// TIA Portal V20 export
VAR_GLOBAL   // PLC tag table "Default tag table"
   BA040AZSDR1_Unwinder1_Interface_AddressIn AT %I5114.0 : "PD_TEL105_IN";
   BA040AZSDR1_Unwinder1_AddressOut AT %Q5114.0 : "PD_TEL105_OUT";
   BA040AZSDR2_Unwinder2_Actor_Interface_AddressIn AT %I5154.0 : "PD_TEL105_IN";
   BA040AZSDR2_Unwinder2_Actor_Interface_AddressOut AT %Q5154.0 : "PD_TEL105_OUT";
   BA040AZSDR5_AnodeMainPnp1AxisX_Actor_Interface_AddressIn AT %I5268.0 : "PD_TEL105_IN";
   BA040AZSDR5_AnodeMainPnp1AxisX_Actor_Interface_AddressOut AT %Q5268.0 : "PD_TEL105_OUT";
   BA040AZSDR6_AnodeMainPnp2AxisX_Actor_Interface_AddressIn AT %I5302.0 : "PD_TEL105_IN";
   BA040AZSDR6_AnodeMainPnp2AxisX_Actor_Interface_AddressOut AT %Q5302.0 : "PD_TEL105_OUT";
   BA040AZSDR7_CathodeMainPnp1AxisX_Actor_Interface_AddressIn AT %I5336.0 : "PD_TEL105_IN";
   BA040AZSDR7_CathodeMainPnp1AxisX_Actor_Interface_AddressOut AT %Q5336.0 : "PD_TEL105_OUT";
   BA040AZSDR8_CathodeMainPnp2AxisX_Actor_Interface_AddressIn AT %I5370.0 : "PD_TEL105_IN";
   BA040AZSDR8_CathodeMainPnp2AxisX_Actor_Interface_AddressOut AT %Q5370.0 : "PD_TEL105_OUT";
   BA040AZSDR9_AnodeMainPnp1AxisY_Actor_Interface_AddressIn AT %I5404.0 : "PD_TEL105_IN";
   BA040AZSDR9_AnodeMainPnp1AxisY_Actor_Interface_AddressOut AT %Q5404.0 : "PD_TEL105_OUT";
   BA040AZSDR10_AnodeMainPnp1AxisZ_Actor_Interface_AddressIn AT %I5438.0 : "PD_TEL105_IN";
   BA040AZSDR10_AnodeMainPnp1AxisZ_Actor_Interface_AddressOut AT %Q5438.0 : "PD_TEL105_OUT";
   BA040AZSDR11_AnodeMainPnp2AxisZ_Actor_Interface_AddressIn AT %I5482.0 : "PD_TEL105_IN";
   BA040AZSDR11_AnodeMainPnp2AxisZ_Actor_Interface_AddressOut AT %Q5482.0 : "PD_TEL105_OUT";
   BA040AZSDR12_CathodeMainPnp2AxisZ_Actor_Interface_AddressIn AT %I5516.0 : "PD_TEL105_IN";
   BA040AZSDR12_CathodeMainPnp2AxisZ_Actor_Interface_AddressOut AT %Q5516.0 : "PD_TEL105_OUT";
   BA040AZSDR13_CathodeMainPnp1AxisX_Actor_Interface_AddressIn AT %I5560.0 : "PD_TEL105_IN";
   BA040AZSDR13_CathodeMainPnp1AxisX_Actor_Interface_AddressOut AT %Q5560.0 : "PD_TEL105_OUT";
   BA040AZSDR14_CathodeMainPnp1AxisZ_Actor_Interface_AddressIn AT %I5604.0 : "PD_TEL105_IN";
   BA040AZSDR14_CathodeMainPnp1AxisZ_Actor_Interface_AddressOut AT %Q5604.0 : "PD_TEL105_OUT";
   BA040AZSDR15_AnodeAlignTableAxisU_Actor_Interface_AddressIn AT %I5648.0 : "PD_TEL105_IN";
   BA040AZSDR15_AnodeAlignTableAxisU_Actor_Interface_AddressOut AT %Q5648.0 : "PD_TEL105_OUT";
   BA040AZSDR16_AnodeAlignTableAxisV_Actor_Interface_AddressIn AT %I5682.0 : "PD_TEL105_IN";
   BA040AZSDR16_AnodeAlignTableAxisV_Actor_Interface_AddressOut AT %Q5682.0 : "PD_TEL105_OUT";
   BA040AZSDR17_AnodeAlignTableAxisW_Actor_Interface_AddressIn AT %I5716.0 : "PD_TEL105_IN";
   BA040AZSDR17_AnodeAlignTableAxisW_Actor_Interface_AddressOut AT %Q5716.0 : "PD_TEL105_OUT";
   BA040AZSDR18_CathodeAlignTableAxisU_Actor_Interface_AddressIn AT %I5750.0 : "PD_TEL105_IN";
   BA040AZSDR18_CathodeAlignTableAxisU_Actor_Interface_AddressOut AT %Q5750.0 : "PD_TEL105_OUT";
   BA040AZSDR19_CathodeAlignTableAxisV_Actor_Interface_AddressIn AT %I5784.0 : "PD_TEL105_IN";
   BA040AZSDR19_CathodeAlignTableAxisV_Actor_Interface_AddressOut AT %Q5784.0 : "PD_TEL105_OUT";
   BA040AZSDR20_CathodeAlignTableAxisW_Actor_Interface_AddressIn AT %I5818.0 : "PD_TEL105_IN";
   BA040AZSDR20_CathodeAlignTableAxisW_Actor_Interface_AddressOut AT %Q5818.0 : "PD_TEL105_OUT";
   BA040AZSDR40_JellyRollWinder1AxisY_Actor_Interface_AddressIn AT %I6588.0 : "PD_TEL105_IN";
   BA040AZSDR40_JellyRollWinder1AxisY_Actor_Interface_AddressOut AT %Q6588.0 : "PD_TEL105_OUT";
   BA040AZSDR41_JellyRollWinder2AxisY_Actor_Interface_AddressIn AT %I6622.0 : "PD_TEL105_IN";
   BA040AZSDR41_JellyRollWinder2AxisY_Actor_Interface_AddressOut AT %Q6622.0 : "PD_TEL105_OUT";
   BA040AZSDR1_UnwinderTopAxisB_Actor_Interface_TorqueDataAddressIn AT %I8000.0 : "PD_TEL750_IN";
   BA040AZSDR1_UnwinderTopAxisB_Actor_Interface_TorqueDataAddressOut AT %Q8000.0 : "PD_TEL750_OUT";
   BA040AZSDR2_UnwinderBottomAxisB_Actor_Interface_TorqueDataAddressIn AT %I8010.0 : "PD_TEL750_IN";
   BA040AZSDR2_UnwinderBottomAxisB_Actor_Interface_TorqueDataAddressOut AT %Q8010.0 : "PD_TEL750_OUT";
   BA040AZSDR4_SepaFeedingRollerAxisB_Actor_Interface_AddressIn AT %I5234.0 : "PD_TEL105_IN";
   BA040AZSDR4_SepaFeedingRollerAxisB_Actor_Interface_AddressOut AT %Q5234.0 : "PD_TEL105_OUT";
   BA040AZSDR4_SepaFeedingRollerAxisB_Actor_Interface_TorqueDataAddressIn AT %I8030.0 : "PD_TEL750_IN";
   BA040AZSDR4_SepaFeedingRollerAxisB_Actor_Interface_TorqueDataAddressOut AT %Q8030.0 : "PD_TEL750_OUT";
   BA040AZSDR21_FinalRollerFrontAxisX_Actor_Interface_AddressIn AT %I5852.0 : "PD_TEL105_IN";
   BA040AZSDR21_FinalRollerFrontAxisX_Actor_Interface_AddressOut AT %Q5852.0 : "PD_TEL105_OUT";
   BA040AZSDR22_FinalRollerRearAxisX_Actor_Interface_AddressIn AT %I5886.0 : "PD_TEL105_IN";
   BA040AZSDR22_FinalRollerRearAxisX_Actor_Interface_AddressOut AT %Q5886.0 : "PD_TEL105_OUT";
   BA040AZSDR23_MendrelAnodeFrontAxisY_Actor_Interface_AddressIn AT %I5920.0 : "PD_TEL105_IN";
   BA040AZSDR23_MendrelAnodeFrontAxisY_Actor_Interface_AddressOut AT %Q5920.0 : "PD_TEL105_OUT";
   BA040AZSDR24_MendrelAnodeFrontAxisZ_Actor_Interface_AddressIn AT %I5954.0 : "PD_TEL105_IN";
   BA040AZSDR24_MendrelAnodeFrontAxisZ_Actor_Interface_AddressOut AT %Q5954.0 : "PD_TEL105_OUT";
   BA040AZSDR25_MendrelAnodeRearAxisY_Actor_Interface_AddressIn AT %I5998.0 : "PD_TEL105_IN";
   BA040AZSDR25_MendrelAnodeRearAxisY_Actor_Interface_AddressOut AT %Q5998.0 : "PD_TEL105_OUT";
   BA040AZSDR26_MendrelAnodeRearAxisZ_Actor_Interface_AddressIn AT %I6032.0 : "PD_TEL105_IN";
   BA040AZSDR26_MendrelAnodeRearAxisZ_Actor_Interface_AddressOut AT %Q6032.0 : "PD_TEL105_OUT";
   BA040AZSDR27_MendrelCathodeFrontAxisY_Actor_Interface_AddressIn AT %I6076.0 : "PD_TEL105_IN";
   BA040AZSDR27_MendrelCathodeFrontAxisY_Actor_Interface_AddressOut AT %Q6076.0 : "PD_TEL105_OUT";
   BA040AZSDR28_MendrelCathodeFrontAxisZ_Actor_Interface_AddressIn AT %I6110.0 : "PD_TEL105_IN";
   BA040AZSDR28_MendrelCathodeFrontAxisZ_Actor_Interface_AddressOut AT %Q6110.0 : "PD_TEL105_OUT";
   BA040AZSDR29_MendrelCathodeRearAxisY_Actor_Interface_AddressIn AT %I6154.0 : "PD_TEL105_IN";
   BA040AZSDR29_MendrelCathodeRearAxisY_Actor_Interface_AddressOut AT %Q6154.0 : "PD_TEL105_OUT";
   BA040AZSDR30_MendrelCathodeRearAxisZ_Actor_Interface_AddressIn AT %I6188.0 : "PD_TEL105_IN";
   BA040AZSDR30_MendrelCathodeRearAxisZ_Actor_Interface_AddressOut AT %Q6188.0 : "PD_TEL105_OUT";
   BA040AZSDR31_StackTableAxisZ_Actor_Interface_AddressIn AT %I6232.0 : "PD_TEL105_IN";
   BA040AZSDR31_StackTableAxisZ_Actor_Interface_AddressOut AT %Q6232.0 : "PD_TEL105_OUT";
   BA040AZSDR32_StackTableOutFrontAxisZ_Actor_Interface_AddressIn AT %I6276.0 : "PD_TEL105_IN";
   BA040AZSDR32_StackTableOutFrontAxisZ_Actor_Interface_AddressOut AT %Q6276.0 : "PD_TEL105_OUT";
   BA040AZSDR33_StackTableOutRearAxisZ_Actor_Interface_AddressIn AT %I6320.0 : "PD_TEL105_IN";
   BA040AZSDR33_StackTableOutRearAxisZ_Actor_Interface_AddressOut AT %Q6320.0 : "PD_TEL105_OUT";
   BA040AZSDR34_SepaClampnCutterAxisX_Actor_Interface_AddressIn AT %I6364.0 : "PD_TEL105_IN";
   BA040AZSDR34_SepaClampnCutterAxisX_Actor_Interface_AddressOut AT %Q6364.0 : "PD_TEL105_OUT";
   BA040AZSDR35_SepaClampnCutterAxisZ_Actor_Interface_AddressIn AT %I6398.0 : "PD_TEL105_IN";
   BA040AZSDR35_SepaClampnCutterAxisZ_Actor_Interface_AddressOut AT %Q6398.0 : "PD_TEL105_OUT";
   BA040AZSDR36_SepaGripperAxisX_Actor_Interface_AddressIn AT %I6442.0 : "PD_TEL105_IN";
   BA040AZSDR36_SepaGripperAxisX_Actor_Interface_AddressOut AT %Q6442.0 : "PD_TEL105_OUT";
   BA040AZSDR37_SepaGripperAxisZ_Actor_Interface_AddressIn AT %I6476.0 : "PD_TEL105_IN";
   BA040AZSDR37_SepaGripperAxisZ_Actor_Interface_AddressOut AT %Q6476.0 : "PD_TEL105_OUT";
   BA040AZSDR38_SepaGripperAxisC_Actor_Interface_AddressIn AT %I6520.0 : "PD_TEL105_IN";
   BA040AZSDR38_SepaGripperAxisC_Actor_Interface_AddressOut AT %Q6520.0 : "PD_TEL105_OUT";
   BA040AZSDR39_JRWinderRearAxisY_Actor_Interface_AddressIn AT %I6554.0 : "PD_TEL105_IN";
   BA040AZSDR39_JRWinderRearAxisY_Actor_Interface_AddressOut AT %Q6554.0 : "PD_TEL105_OUT";
   BA040AZSDR3_CompensatorAxisX_Actor_Interface_AddressIn AT %I5194.0 : "PD_TEL105_IN";
   BA040AZSDR3_CompensatorAxisX_Actor_Interface_AddressOut AT %Q5194.0 : "PD_TEL105_OUT";
   BA040AZSDR3_CompensatorAxisX_Actor_Interface_TorqueDataAddressIn AT %I8020.0 : "PD_TEL750_IN";
   BA040AZSDR3_CompensatorAxisX_Actor_Interface_TorqueDataAddressOut AT %Q8020.0 : "PD_TEL750_OUT";
   BA040AZSDR39_JRWinderRearAxisY_Actor_Interface_TorqueDataAddressIn AT %I8380.0 : "PD_TEL750_IN";
   BA040AZSDR39_JRWinderRearAxisY_Actor_Interface_TorqueDataAddressOut AT %Q8380.0 : "PD_TEL750_OUT";
   BA040AZSDR5_AnodeMainPnp1AxisX_Actor_Interface_TorqueDataAddressIn AT %I8040.0 : "PD_TEL750_IN";
   BA040AZSDR5_AnodeMainPnp1AxisX_Actor_Interface_TorqueDataAddressOut AT %Q8040.0 : "PD_TEL750_OUT";
   BA040AZSDR6_AnodeMainPnp2AxisX_Actor_Interface_TorqueDataAddressIn AT %I8050.0 : "PD_TEL750_IN";
   BA040AZSDR6_AnodeMainPnp2AxisX_Actor_Interface_TorqueDataAddressOut AT %Q8050.0 : "PD_TEL750_OUT";
   BA040AZSDR11_AnodeMainPnp1AxisY_Actor_Interface_TorqueDataAddressIn AT %I8100.0 : "PD_TEL750_IN";
   BA040AZSDR11_AnodeMainPnp1AxisY_Actor_Interface_TorqueDataAddressOut AT %Q8100.0 : "PD_TEL750_OUT";
   BA040AZSDR12_AnodeMainPnp1AxisZ_Actor_Interface_TorqueDataAddressIn AT %I8110.0 : "PD_TEL750_IN";
   BA040AZSDR12_AnodeMainPnp1AxisZ_Actor_Interface_TorqueDataAddressOut AT %Q8110.0 : "PD_TEL750_OUT";
   BA040AZSDR14_AnodeMainPnp2AxisZ_Actor_Interface_TorqueDataAddressIn AT %I8130.0 : "PD_TEL750_IN";
   BA040AZSDR14_AnodeMainPnp2AxisZ_Actor_Interface_TorqueDataAddressOut AT %Q8130.0 : "PD_TEL750_OUT";
   BA040AZSDR15_AnodeAlignTableAxisX_Actor_Interface_TorqueDataAddressIn AT %I8140.0 : "PD_TEL750_IN";
   BA040AZSDR15_AnodeAlignTableAxisX_Actor_Interface_TorqueDataAddressOut AT %Q8140.0 : "PD_TEL750_OUT";
   BA040AZSDR16_AnodeAlignTableAxisY1_Actor_Interface_TorqueDataAddressIn AT %I8150.0 : "PD_TEL750_IN";
   BA040AZSDR16_AnodeAlignTableAxisY1_Actor_Interface_TorqueDataAddressOut AT %Q8150.0 : "PD_TEL750_OUT";
   BA040AZSDR17_AnodeAlignTableAxisY2_Actor_Interface_TorqueDataAddressIn AT %I8160.0 : "PD_TEL750_IN";
   BA040AZSDR17_AnodeAlignTableAxisY2_Actor_Interface_TorqueDataAddressOut AT %Q8160.0 : "PD_TEL750_OUT";
   BA040AZSDR7_CathodeMainPnp1AxisX_Actor_Interface_TorqueDataAddressIn AT %I8060.0 : "PD_TEL750_IN";
   BA040AZSDR7_CathodeMainPnp1AxisX_Actor_Interface_TorqueDataAddressOut AT %Q8060.0 : "PD_TEL750_OUT";
   BA040AZSDR8_CathodeMainPnp2AxisX_Actor_Interface_TorqueDataAddressIn AT %I8070.0 : "PD_TEL750_IN";
   BA040AZSDR8_CathodeMainPnp2AxisX_Actor_Interface_TorqueDataAddressOut AT %Q8070.0 : "PD_TEL750_OUT";
   BA040AZSDR9_CathodeMainPnp1AxisY_Actor_Interface_TorqueDataAddressIn AT %I8080.0 : "PD_TEL750_IN";
   BA040AZSDR9_CathodeMainPnp1AxisY_Actor_Interface_TorqueDataAddressOut AT %Q8080.0 : "PD_TEL750_OUT";
   BA040AZSDR10_CathodeMainPnp1AxisZ_Actor_Interface_TorqueDataAddressIn AT %I8090.0 : "PD_TEL750_IN";
   BA040AZSDR10_CathodeMainPnp1AxisZ_Actor_Interface_TorqueDataAddressOut AT %Q8090.0 : "PD_TEL750_OUT";
   BA040AZSDR13_CathodeMainPnp2AxisZ_Actor_Interface_TorqueDataAddressIn AT %I8120.0 : "PD_TEL750_IN";
   BA040AZSDR13_CathodeMainPnp2AxisZ_Actor_Interface_TorqueDataAddressOut AT %Q8120.0 : "PD_TEL750_OUT";
   BA040AZSDR18_CathodeAlignTableAxisX_Actor_Interface_TorqueDataAddressIn AT %I8170.0 : "PD_TEL750_IN";
   BA040AZSDR18_CathodeAlignTableAxisX_Actor_Interface_TorqueDataAddressOut AT %Q8170.0 : "PD_TEL750_OUT";
   BA040AZSDR19_CathodeAlignTableAxisY1_Actor_Interface_TorqueDataAddressIn AT %I8180.0 : "PD_TEL750_IN";
   BA040AZSDR19_CathodeAlignTableAxisY1_Actor_Interface_TorqueDataAddressOut AT %Q8180.0 : "PD_TEL750_OUT";
   BA040AZSDR20_CathodeAlignTableAxisY2_Actor_Interface_TorqueDataAddressIn AT %I8190.0 : "PD_TEL750_IN";
   BA040AZSDR20_CathodeAlignTableAxisY2_Actor_Interface_TorqueDataAddressOut AT %Q8190.0 : "PD_TEL750_OUT";
   BA040AZSDR21_FinalRollerFrontAxisX_Actor_Interface_TorqueDataAddressIn AT %I8200.0 : "PD_TEL750_IN";
   BA040AZSDR21_FinalRollerFrontAxisX_Actor_Interface_TorqueDataAddressOut AT %Q8200.0 : "PD_TEL750_OUT";
   BA040AZSDR22_FinalRollerRearAxisX_Actor_Interface_TorqueDataAddressIn AT %I8210.0 : "PD_TEL750_IN";
   BA040AZSDR22_FinalRollerRearAxisX_Actor_Interface_TorqueDataAddressOut AT %Q8210.0 : "PD_TEL750_OUT";
   BA040AZSDR23_MendrelAnodeFrontAxisY_Actor_Interface_TorqueDataAddressIn AT %I8220.0 : "PD_TEL750_IN";
   BA040AZSDR23_MendrelAnodeFrontAxisY_Actor_Interface_TorqueDataAddressOut AT %Q8220.0 : "PD_TEL750_OUT";
   BA040AZSDR24_MendrelAnodeFrontAxisZ_Actor_Interface_TorqueDataAddressIn AT %I8230.0 : "PD_TEL750_IN";
   BA040AZSDR24_MendrelAnodeFrontAxisZ_Actor_Interface_TorqueDataAddressOut AT %Q8230.0 : "PD_TEL750_OUT";
   BA040AZSDR25_MendrelAnodeRearAxisY_Actor_Interface_TorqueDataAddressIn AT %I8240.0 : "PD_TEL750_IN";
   BA040AZSDR25_MendrelAnodeRearAxisY_Actor_Interface_TorqueDataAddressOut AT %Q8240.0 : "PD_TEL750_OUT";
   BA040AZSDR26_MendrelAnodeRearAxisZ_Actor_Interface_TorqueDataAddressIn AT %I8250.0 : "PD_TEL750_IN";
   BA040AZSDR26_MendrelAnodeRearAxisZ_Actor_Interface_TorqueDataAddressOut AT %Q8250.0 : "PD_TEL750_OUT";
   BA040AZSDR27_MendrelCathodeFrontAxisY_Actor_Interface_TorqueDataAddressIn AT %I8260.0 : "PD_TEL750_IN";
   BA040AZSDR27_MendrelCathodeFrontAxisY_Actor_Interface_TorqueDataAddressOut AT %Q8260.0 : "PD_TEL750_OUT";
   BA040AZSDR28_MendrelCathodeFrontAxisZ_Actor_Interface_TorqueDataAddressIn AT %I8270.0 : "PD_TEL750_IN";
   BA040AZSDR28_MendrelCathodeFrontAxisZ_Actor_Interface_TorqueDataAddressOut AT %Q8270.0 : "PD_TEL750_OUT";
   BA040AZSDR29_MendrelCathodeRearAxisY_Actor_Interface_TorqueDataAddressIn AT %I8280.0 : "PD_TEL750_IN";
   BA040AZSDR29_MendrelCathodeRearAxisY_Actor_Interface_TorqueDataAddressOut AT %Q8280.0 : "PD_TEL750_OUT";
   BA040AZSDR30_MendrelCathodeRearAxisZ_Actor_Interface_TorqueDataAddressIn AT %I8290.0 : "PD_TEL750_IN";
   BA040AZSDR30_MendrelCathodeRearAxisZ_Actor_Interface_TorqueDataAddressOut AT %Q8290.0 : "PD_TEL750_OUT";
   BA040AZSDR31_StackTableAxisZ_Actor_Interface_TorqueDataAddressIn AT %I8300.0 : "PD_TEL750_IN";
   BA040AZSDR31_StackTableAxisZ_Actor_Interface_TorqueDataAddressOut AT %Q8300.0 : "PD_TEL750_OUT";
   BA040AZSDR32_StackTableOutFrontAxisZ_Actor_Interface_TorqueDataAddressIn AT %I8310.0 : "PD_TEL750_IN";
   BA040AZSDR32_StackTableOutFrontAxisZ_Actor_Interface_TorqueDataAddressOut AT %Q8310.0 : "PD_TEL750_OUT";
   BA040AZSDR33_StackTableOutRearAxisZ_Actor_Interface_TorqueDataAddressIn AT %I8320.0 : "PD_TEL750_IN";
   BA040AZSDR33_StackTableOutRearAxisZ_Actor_Interface_TorqueDataAddressOut AT %Q8320.0 : "PD_TEL750_OUT";
   BA040AZSDR34_SepaClampnCutterAxisX_Actor_Interface_TorqueDataAddressIn AT %I8330.0 : "PD_TEL750_IN";
   BA040AZSDR34_SepaClampnCutterAxisX_Actor_Interface_TorqueDataAddressOut AT %Q8330.0 : "PD_TEL750_OUT";
   BA040AZSDR35_SepaClampnCutterAxisZ_Actor_Interface_TorqueDataAddressIn AT %I8340.0 : "PD_TEL750_IN";
   BA040AZSDR35_SepaClampnCutterAxisZ_Actor_Interface_TorqueDataAddressOut AT %Q8340.0 : "PD_TEL750_OUT";
   BA040AZSDR36_SepaGripperAxisX_Actor_Interface_TorqueDataAddressIn AT %I8350.0 : "PD_TEL750_IN";
   BA040AZSDR36_SepaGripperAxisX_Actor_Interface_TorqueDataAddressOut AT %Q8350.0 : "PD_TEL750_OUT";
   BA040AZSDR37_SepaGripperAxisZ_Actor_Interface_TorqueDataAddressIn AT %I8360.0 : "PD_TEL750_IN";
   BA040AZSDR37_SepaGripperAxisZ_Actor_Interface_TorqueDataAddressOut AT %Q8360.0 : "PD_TEL750_OUT";
   BA040AZSDR38_SepaGripperAxisC_Actor_Interface_TorqueDataAddressIn AT %I8370.0 : "PD_TEL750_IN";
   BA040AZSDR38_SepaGripperAxisC_Actor_Interface_TorqueDataAddressOut AT %Q8370.0 : "PD_TEL750_OUT";
   BA040AZSDR40_JRWinderFrontAxisY_Actor_Interface_TorqueDataAddressIn AT %I8390.0 : "PD_TEL750_IN";
   BA040AZSDR40_JRWinderFrontAxisY_Actor_Interface_TorqueDataAddressOut AT %Q8390.0 : "PD_TEL750_OUT";
   BA040AZSDR41_JRWinderAxisB_Actor_Interface_TorqueDataAddressIn AT %I8440.0 : "PD_TEL750_IN";
   BA040AZSDR41_JRWinderAxisB_Actor_Interface_TorqueDataAddressOut AT %Q8440.0 : "PD_TEL750_OUT";
   "BA040AZSSP512.00" AT %Q3550.0 : Bool;   // UNWINDER EPCC04 INTERKOCK
END_VAR
